// Mitsubishi GX Works2 project: 0715로테이션쉬프트1   PLC: Q02/Q02H

PROGRAM MAIN
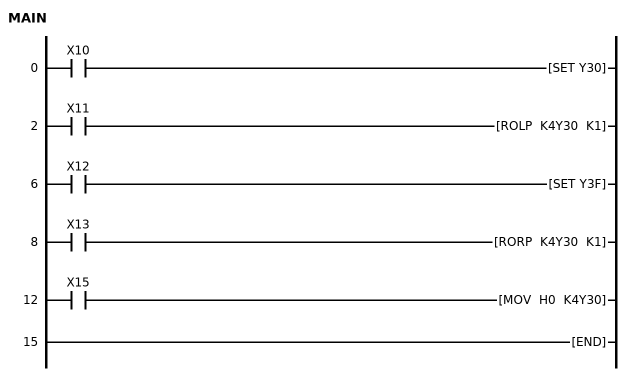
0     LD      X10
      SET     Y30
2     LD      X11
      ROLP    K4Y30 K1
6     LD      X12
      SET     Y3F
8     LD      X13
      RORP    K4Y30 K1
12    LD      X15
      MOV     H0 K4Y30
15    END
END_PROGRAM
